FUNCTION Mapping_ModbusReadRegisters
VAR_INPUT
	Read_Struct : POINTER TO ScaledModRead;
	ToSLCVariables : POINTER TO EtherCAT_Monitor_Variables;
	ToSLCStatus : POINTER TO EtherCAT_Stat_Variables;
	
END_VAR
VAR
END_VAR

//Variables
	//Status Parameter
		ToSLCStatus^.Status := Read_Struct^.fbOpMode;				// This data block is for send modbus FLC-SLC
	//Battery parameters
		ToSLCVariables^.BatSoc := Read_Struct^.BatSoc;
		//ToSLCVariables^.BatSocUpLim := Read_Struct^.BatSocUpLimit;
		//ToSLCVariables^.BatSocLowLim := Read_Struct^.BatSocLowLimit;
	//Active and Reactive Power Reference
		ToSLCVariables^.TotW := Read_Struct^.TotW;
		ToSLCVariables^.TotVAr := Read_Struct^.TotVAr;
	//Grid Frequency
		ToSLCVariables^.GridFre := Read_Struct^.GridFre;
	//Grid Currents RMS
		ToSLCVariables^.Irmsa := Read_Struct^.Irmsa;
		ToSLCVariables^.Irmsb := Read_Struct^.Irmsb;
		ToSLCVariables^.Irmsc := Read_Struct^.Irmsc;
	//Grid Voltages RMS
		ToSLCVariables^.Vrmsa := Read_Struct^.Vrmsa;
		ToSLCVariables^.Vrmsb := Read_Struct^.Vrmsb;
		ToSLCVariables^.Vrmsc := Read_Struct^.Vrmsc;
	//HeartBeat reading
		ToSLCStatus^.HeartBeat := Read_Struct^.HeartBeat;

END_FUNCTION

(* stored: Version 1.1.0.1, ProductVersion 3.1.4024.2
   POU Mapping_ModbusReadRegisters: Id {9fd71e59-685d-4706-af32-6ef0044453b3}, SpecialFunc None *)
